// TwinCAT 3 PLC project LCLSGeneral
// Title: LCLS General-jozamudi
// Company: SLAC
// Author: Alex Wallace
// ProjectVersion: 0.0.0
// Description: Generally useful POUs: - Logger - FB diagnostics - EtherCAT diagnostic
// ProgramVersion: 3.1.4020.2
// libraries:
//   Tc2_EtherCAT, * (Beckhoff Automation GmbH)
//   Tc2_IoFunctions, * (Beckhoff Automation GmbH)
//   Tc2_ModbusSrv, * (Beckhoff Automation GmbH)
//   Tc2_SerialCom, * (Beckhoff Automation GmbH)
//   Tc2_Standard, * (Beckhoff Automation GmbH)
//   Tc2_System, * (Beckhoff Automation GmbH)
//   Tc2_TcpIp, * (Beckhoff Automation GmbH)
//   Tc2_Utilities, * (Beckhoff Automation GmbH)
//   Tc3_EventLogger, * (Beckhoff Automation GmbH)
//   Tc3_JsonXml, * (Beckhoff Automation GmbH)
//   Tc3_Module, * (Beckhoff Automation GmbH)
//   TcUnit, * (www.tcunit.org)
// project tree:
//   Data types/EPICS/ ST_EpicsMotorMSTA.TcDUT (not stored)
//   Data types/Misc/ ST_EcDevice.TcDUT (not stored), ST_FbDiagnostics.TcDUT (not stored), ST_System.TcDUT (not stored)
//   DUT/ DUT_EPS.TcDUT
//   GVLs/ GeneralConstants.TcGVL (not stored), DefaultGlobals.TcGVL (not stored), Global_Variables_EtherCAT.TcGVL (not stored)
//   POUs/Data/ FB_BasicStats.TcPOU (not stored), FB_DataBuffer.TcPOU (not stored), FB_EpicsCentroidMonitor.TcPOU (not stored), FB_EpicsMotorMonitor.TcPOU (not stored), FB_LREALBuffer.TcPOU (not stored), FB_LREALFromEPICS.TcPOU (not stored), FB_STRINGFromEPICS.TcPOU (not stored), FB_TimeStampBuffer.TcPOU (not stored), FB_TimeStampBufferGlobal.TcPOU (not stored)
//   POUs/Data/Tests/ FB_Test_EpicsCentroidMonitor.TcPOU (not stored), FB_Test_EpicsMotorMonitor.TcPOU (not stored)
//   POUs/Diagnostics/DUT/ E_EcatDiagState.TcDUT (not stored), E_EcCommState.TcDUT (not stored), ST_EcMasterDevState.TcDUT (not stored), ST_PortAddr.TcDUT (not stored), ST_SlaveState.TcDUT (not stored), ST_SlaveStateInfo.TcDUT (not stored), ST_SlaveStateInfoScanned.TcDUT (not stored), ST_TopologyData.TcDUT (not stored)
//   POUs/Diagnostics/ FB_EcatDiagWrapper.TcPOU (not stored), FB_EtherCATDiag.TcPOU (not stored), FB_EtherCATFrameDiag.TcPOU (not stored)
//   POUs/EPS/ FB_EPS.TcPOU
//   POUs/Functions/ FB_EcatDiag.TcPOU (not stored), FB_Index.TcPOU (not stored), FB_UnixTimeStamp.TcPOU (not stored), FB_UnixTimeStampGlobal.TcPOU (not stored), FB_XKoyoPLCModbus.TcPOU (not stored), F_ConvertTicksToUnixTimestamp.TcPOU (not stored), TIME_TO_100NS.TcPOU (not stored)
//   POUs/Hardware/ FB_AnalogOutput.TcPOU (not stored), FB_AnalogInput.TcPOU (not stored), FB_CoE_FastRead.TcPOU (not stored), FB_EL6_Com.TcPOU (not stored), FB_GetPLCHostname.TcPOU (not stored), FB_GetPLCIPAddress.TcPOU (not stored), FB_LED.TcPOU (not stored), FB_ThermoCouple.TcPOU (not stored), FB_TempSensor.TcPOU (not stored)
//   POUs/Logger/DUTs/ E_LogEventType_WC.TcDUT (not stored), ST_LoggingEventInfo_WC.TcDUT (not stored), ST_PendingEvent.TcDUT (not stored), E_Subsystem.TcDUT (not stored)
//   POUs/Logger/ FB_Listener.TcPOU (not stored), FB_LogHandler.TcPOU (not stored), FB_LogMessage.TcPOU (not stored), F_SendUDPMessage.TcPOU (not stored), GVL_Logger.TcGVL (not stored), SYSTEM_TIME_TO_RFC3339.TcPOU (not stored)
//   POUs/Logger/Tests/ FB_CircuitBreaker_Test.TcPOU (not stored), ResetCircuitBreakerGlobals.TcPOU (not stored)
//   POUs/ RUN_TESTS.TcPOU (not stored)
//   / Task_3.TcTTO (not stored)
// real-time tasks:
//   TASK Task 3: cycle T#10ms, priority 1, ADS port 350

// ---- DUT/DUT_EPS.TcDUT
TYPE DUT_EPS :
STRUCT
	// Contains EPS flags
    {attribute 'pytmc' := '
        pv: EPS:nFlags
        io: io
        field: DESC Contains EPS flags
    '}
	nFlags: UDINT:=0;
    
    // Desciption of values nFlags contains
	{attribute 'pytmc' := '
		pv:EPS:sDesc
		io: io
		field: DESC of nFlag variable
	'}
	sFlagDesc:  STRING;
	
	// Number of bits used in nFlags
	{attribute 'pytmc' := '
		pv: EPS:nNBitUsed
		io: io
		field: DESC number of bits used
	'}
	nBitsUsed: BYTE;
	
	// Name to use for log messages.
    {attribute 'pytmc' := '
        pv: EPS:sMessage
        io: i
        field: DESC Message from EPS to usr
    '}
    sMessage: STRING;
END_STRUCT
END_TYPE

// ---- POUs/EPS/FB_EPS.TcPOU
FUNCTION_BLOCK FB_EPS
VAR_IN_OUT
    eps : DUT_EPS;
END_VAR
VAR_OUTPUT
END_VAR
VAR 
END_VAR

METHOD setBit : BOOL
VAR_INPUT
    nBits : BYTE;
	bValue : BOOL;
END_VAR
VAR
    nMask : UDINT := 1;
	nBitValue : UDINT := 0;
END_VAR
nMask := SHL(nMask, nBits);
nBitValue := SHR((nMask AND eps.nFlags), nBits);

IF (TO_BOOL(nBitValue)) <> bValue THEN
	eps.nFlags := eps.nFlags XOR nmask;
END_IF
END_METHOD

METHOD setBitsUsed : BOOL
VAR_INPUT
	bitsUsed : BYTE;
END_VAR
eps.nBitsUsed := bitsUsed;
END_METHOD

METHOD setDescription : BOOL
VAR_INPUT
	desciption : STRING;
END_VAR
eps.sFlagDesc := desciption;
END_METHOD

METHOD setMessage : BOOL
VAR_INPUT
    message : STRING;
END_VAR
eps.sMessage := message;
END_METHOD

END_FUNCTION_BLOCK
